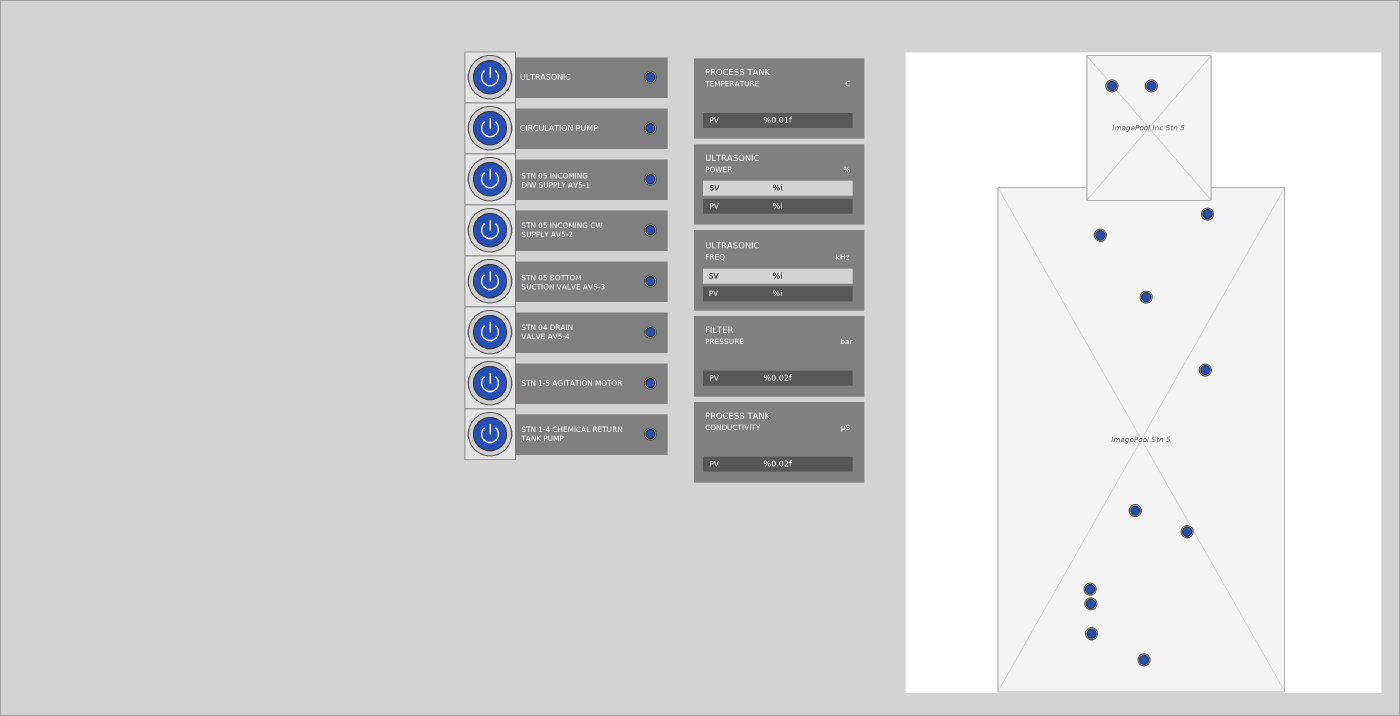
VISUALIZATION Manual_Station05  // 1920x983
    Rectangle (0,0 1920x983)
    Rectangle (1242,72 652x879)
    Image (1368,257 394x693), image: ImagePool.Stn 5
    RoundedRectangle (676,79 239x55)
    Label (710,98 163x16), "ULTRASONIC"
    Lamp1 (882,96 20x20), variable: ARdsMAP_HmiVariableStn[5].bProTankUsBtm_IND, style: Lamp-Lamp1-Blue
    PowerSwitch (637,71 70x70), variable: ARdsMAP_HmiVariableStn[5].bProTankUsBtm_PB, behaviour: TOGGLE, style: Switch-PowerSwitch-Blue
    RoundedRectangle (684,149 231x55)
    Label (710,168 151x16), "CIRCULATION PUMP"
    Lamp1 (882,166 20x20), variable: ARdsMAP_HmiVariableStn[5].bProTankPump_IND, style: Lamp-Lamp1-Blue
    PowerSwitch (637,141 70x70), variable: ARdsMAP_HmiVariableStn[5].bProTankPump_PB, behaviour: TOGGLE, style: Switch-PowerSwitch-Blue
    RoundedRectangle (952,80 233x110)
    Label (964,91 150x16), "PROCESS TANK"
    Label (964,104 99x22), "TEMPERATURE"
    Label (1140,104 29x22), "C"
    Rectangle (964,155 205x20), "%0.01f", text variable: ARrStnTempPV[5]
    Label (970,154 22x22), "PV"
    Group (952,198 233x110)
        RoundedRectangle (0,0 233x110)
        Label (12,11 150x16), "ULTRASONIC"
        Label (12,24 99x22), "POWER"
        Label (188,24 29x22), "%"
        Rectangle (12,50 205x20), "%i", text variable: ARiStnManualUSBtmAsv[5]
            OnMouseDown: write the text variable via VisuDialogs.Numpad, min 10, max 100
        Label (18,49 22x22), "SV"
        Rectangle (12,75 205x20), "%i", text variable: ARiStnUSBtmAPv[5]
        Label (18,74 22x22), "PV"
    Group (952,434 233x110)
        RoundedRectangle (0,0 233x110)
        Label (12,11 150x16), "FILTER"
        Label (12,24 99x22), "PRESSURE"
        Label (188,24 32x22), "bar"
        Rectangle (12,75 205x20), "%0.02f", text variable: ARrStnFilterPressurePV[5]
        Label (18,74 22x22), "PV"
    Group (952,552 233x110)
        RoundedRectangle (0,0 233x110)
        Label (12,11 150x16), "PROCESS TANK"
        Label (12,24 99x22), "CONDUCTIVITY"
        Label (188,24 29x22), "μS"
        Label (18,49 22x22)
        Rectangle (12,75 205x20), "%0.02f", text variable: ARrStnConductivityPV[5]
        Label (18,74 22x22), "PV"
    Group (952,316 233x110)
        RoundedRectangle (0,0 233x110)
        Label (12,26 99x22), "FREQ"
        Label (12,13 150x16), "ULTRASONIC"
        Label (187,26 29x22), "kHz"
        Rectangle (12,77 205x20), "%i", text variable: ARiStnUSBtmAFreqPv[5]
        Label (17,76 22x22), "PV"
        Rectangle (12,53 205x20), "%i", text variable: DSWeberEnclosure[2].DSWeberGenerator[3].DSWeberMulFreqSwitching.iFreqOutput_TS
            tap DSWeberEnclosure[2].DSWeberGenerator[3].DSWeberMulFreqSwitching.bFreqSwitchingPB_TS
        Label (17,52 22x22), "SV"
    RoundedRectangle (684,289 231x55)
    Label (712,298 160x36), "STN 05 INCOMING CW SUPPLY AV5-2"
    Lamp1 (882,306 20x20), variable: ARdsMAP_HmiVariableStn[5].bValve02_IND, style: Lamp-Lamp1-Blue
    PowerSwitch (637,281 70x70), variable: ARdsMAP_HmiVariableStn[5].bValve02_PB, behaviour: TOGGLE, style: Switch-PowerSwitch-Blue
    RoundedRectangle (684,429 231x55)
    Label (712,438 160x36), "STN 04 DRAIN VALVE AV5-4"
    Lamp1 (882,446 20x20), variable: ARdsMAP_HmiVariableStn[5].bValve04_IND, style: Lamp-Lamp1-Blue
    PowerSwitch (637,421 70x70), variable: ARdsMAP_HmiVariableStn[5].bValve04_PB, behaviour: TOGGLE, style: Switch-PowerSwitch-Blue
    RoundedRectangle (684,359 231x55)
    Lamp1 (882,376 20x20), variable: ARdsMAP_HmiVariableStn[5].bValve03_IND, style: Lamp-Lamp1-Blue
    PowerSwitch (637,351 70x70), variable: ARdsMAP_HmiVariableStn[5].bValve03_PB, behaviour: TOGGLE, style: Switch-PowerSwitch-Blue
    Label (712,370 151x36), "STN 05 BOTTOM SUCTION VALVE AV5-3"
    RoundedRectangle (684,219 231x55)
    Lamp1 (882,236 20x20), variable: ARdsMAP_HmiVariableStn[5].bValve01_IND, style: Lamp-Lamp1-Blue
    PowerSwitch (637,211 70x70), variable: ARdsMAP_HmiVariableStn[5].bValve01_PB, behaviour: TOGGLE, style: Switch-PowerSwitch-Blue
    Label (712,230 151x36), "STN 05 INCOMING DIW SUPPLY AV5-1"
    RoundedRectangle (684,499 231x55)
    Label (712,508 160x36), "STN 1-5 AGITATION MOTOR"
    Lamp1 (882,516 20x20), variable: ARdsMAP_HmiVariableGeneral.bProTankAgitationMotor_IND, style: Lamp-Lamp1-Blue
    PowerSwitch (637,491 70x70), variable: ARdsMAP_HmiVariableGeneral.bProTankAgitationMotor_PB, behaviour: TOGGLE, style: Switch-PowerSwitch-Blue
    Lamp1 (1562,398 20x20), variable: ARdsMAP_HmiVariableStn[5].bProTankUsBtm_IND, style: Lamp-Lamp1-Blue
    Lamp1 (1547,691 20x20), variable: ARdsMAP_HmiVariableStn[5].bProTankPump_IND, style: Lamp-Lamp1-Blue
    Lamp1 (1618,720 20x20), variable: ARdsMAP_HmiVariableStn[5].bValve04_IND, style: Lamp-Lamp1-Blue
    Lamp1 (1643,498 20x20), variable: ARdsMAP_HmiVariableStn[5].bValve03_IND, style: Lamp-Lamp1-Blue
    Lamp1 (1499,313 20x20), variable: ARdsMAP_HmiVariableStn[5].bProcessTankMinLevel_IND, style: Lamp-Lamp1-Blue
    Lamp1 (1646,284 20x20), variable: ARdsMAP_HmiVariableStn[5].bOverflowMaxLevel_IND, style: Lamp-Lamp1-Blue
    Lamp1 (1487,860 20x20), variable: ARdsMAP_HmiVariableStn[5].bSubTankMinLevel_IND, style: Lamp-Lamp1-Blue
    Lamp1 (1486,819 20x20), variable: ARdsMAP_HmiVariableStn[5].bSubTankRegLevel_IND, style: Lamp-Lamp1-Blue
    Lamp1 (1485,799 20x20), variable: ARdsMAP_HmiVariableStn[5].bSubTankMaxLevel_IND, style: Lamp-Lamp1-Blue
    RoundedRectangle (684,569 231x55)
    Label (712,578 170x36), "STN 1-4 CHEMICAL RETURN TANK PUMP"
    Lamp1 (882,586 20x20), variable: ARdsMAP_HmiVariableGeneral.bProTankPump_IND, style: Lamp-Lamp1-Blue
    PowerSwitch (637,561 70x70), variable: ARdsMAP_HmiVariableGeneral.bProTankPump_PB, behaviour: TOGGLE, style: Switch-PowerSwitch-Blue
    Lamp1 (1559,896 20x20), variable: ARdsMAP_HmiVariableGeneral.bProTankPump_IND, style: Lamp-Lamp1-Blue
    Image (1490,76 171x199), image: ImagePool.Inc Stn 5
    Lamp1 (1515,108 20x20), variable: ARdsMAP_HmiVariableStn[5].bValve01_IND, style: Lamp-Lamp1-Blue
    Lamp1 (1569,108 20x20), variable: ARdsMAP_HmiVariableStn[5].bValve02_IND, style: Lamp-Lamp1-Blue
END_VISUALIZATION

(* stored: Version 1.1.0.1, ProductVersion 3.1.4024.12
   Visu Manual_Station05: Id {4b5bff83-b2c8-4933-af5a-7a3a2f819472} *)
